// TIA Portal V16 export
// export: Created 2022-11-14T17:35:50.178922Z, ExportSetting WithDefaults, DisplayName Totally Integrated Automation Portal, DisplayVersion V16, DisplayName TIA Portal Version Control Interface, DisplayVersion V16, DisplayName TIA Portal Openness, DisplayVersion V16, DisplayName STEP 7 Professional, DisplayVersion V16, DisplayName STEP 7 Safety, DisplayVersion V16, DisplayName WinCC Advanced, DisplayVersion V16
DATA_BLOCK "DB252_ProgramGreyBar"   // DB252
{ S7_Optimized_Access := 'FALSE' }
VERSION : 0.1
// stored: AutoNumber false, IsOnlyStoredInLoadMemory false, IsWriteProtectedInAS false
   VAR RETAIN
      Height { ExternalAccessible := 'False'; ExternalVisible := 'False'; ExternalWritable := 'False'; S7_SetPoint := 'True'} : Array[1..13] of "ProgramDataGreyBar";
   END_VAR
BEGIN
   Height[1..2].Overlap := 0;
   Height[3..4].Overlap := 100;
   Height[5..13].Overlap := 0;
   Height[1].Height := 130;
   Height[2].Height := 50;
   Height[3].Height := -50;
   Height[4].Height := 100;
   Height[5].Height := 50;
   Height[6..13].Height := 0;
   Height[1..2].Landmark := FALSE;
   Height[3].Landmark := TRUE;
   Height[4..13].Landmark := FALSE;
   Height[1..13].Lifter := FALSE;
   Height[1..13].SpareBit1 := FALSE;
   Height[1..5].Airblower := TRUE;
   Height[6..13].Airblower := FALSE;
   Height[1..4].NextStep := TRUE;
   Height[5..13].NextStep := FALSE;
   Height[1..4].PressureP := TRUE;
   Height[5..13].PressureP := FALSE;
   Height[1..13].SpareByte1 := 16#00;
   Height[1..2].Revolution := 1;
   Height[3].Revolution := 2;
   Height[4].Revolution := 3;
   Height[5].Revolution := 1;
   Height[6..13].Revolution := 0;
   Height[1..3].RopeUnitUpper := 16#01;
   Height[4].RopeUnitUpper := 16#02;
   Height[5].RopeUnitUpper := 16#01;
   Height[6..13].RopeUnitUpper := 16#00;
   Height[1..3].RopeUnitLower := 16#01;
   Height[4].RopeUnitLower := 16#02;
   Height[5].RopeUnitLower := 16#01;
   Height[6..13].RopeUnitLower := 16#00;
   Height[1].FilmForce := 5;
   Height[2].FilmForce := 20;
   Height[3..5].FilmForce := 30;
   Height[6..13].FilmForce := 0;
   Height[1..5].FilmPrestretch := 200;
   Height[6..13].FilmPrestretch := 0;
   Height[1..13].SpareWord1 := 0;
   Height[1..13].SpareWord2 := 0;
   Height[1..13].SpareWord3 := 0;
   Height[1..2].SpareWord4 := 0;
   Height[3].SpareWord4 := 380;
   Height[4..13].SpareWord4 := 0;
   Height[1..2].SpareWord5 := 0;
   Height[3].SpareWord5 := 2800;
   Height[4..13].SpareWord5 := 0;
   Height[1..13].SpareWord6 := 0;
END_DATA_BLOCK
